// TIA Portal V20 export
DATA_BLOCK "DI3"   // DB280
// stored: MemoryReserve 100
   VAR
      "EQUIPMENT LED POWER TRIPPED E6780CB" : Bool;
      "MOTOR POWER MC COIL POWER TRIPPED E6786CB" : Bool;
      "SAFETY POWER SMPS DC OK E6804PWS" : Bool;
      "SAFETY DC POWER TRIPPED E6808CB" : Bool;
      "ET200SP I/O SAFETY POWER TRIPPED E6816CB" : Bool;
      "JUNCTION BOX CONTROL POWER TRIPPED E6836CB" : Bool;
      "ET200ECO PN-SAFETY-1 POWER TRIPPED E6856CB" : Bool;
      SPARE1 : Bool;
      SPARE2 : Bool;
      SPARE3 : Bool;
      SPARE4 : Bool;
      SPARE5 : Bool;
      SPARE6 : Bool;
      SPARE7 : Bool;
      SPARE8 : Bool;
      SPARE9 : Bool;
      SPARE10 : Bool;
      SPARE11 : Bool;
      SPARE12 : Bool;
      SPARE13 : Bool;
      SPARE14 : Bool;
      SPARE15 : Bool;
      SPARE16 : Bool;
      SPARE17 : Bool;
      SPARE18 : Bool;
      SPARE19 : Bool;
      SPARE20 : Bool;
      SPARE21 : Bool;
      SPARE22 : Bool;
      SPARE23 : Bool;
      SPARE24 : Bool;
      SPARE25 : Bool;
   END_VAR
BEGIN
END_DATA_BLOCK
